PROGRAM MAIN
VAR
	bStart 						: BOOL;
	bEnable 					: BOOL;
	bDisable 					: BOOL;
	bReset 						: BOOL;
	bStop						: BOOL;
	nCase 						: UINT;
	nDemoSequenceState			: UINT;
	
	fbMover						: MC_PlanarMover;
	cmdFB						: MC_PlanarFeedback;
	stMoverState				: MC_PLANAR_STATE;
	stMoverPosition				: ARRAY[1..5] OF PositionXYC;
	fbDnyMove					: DynamicConstraint_PathXY;
	fbDnyRotate					: DynamicConstraint_Coordinates;
	stMoveCOptions				: ST_MoveCOptions;
	
	// Homing
	fbHomeATasks				: FB_TaskMoveA_tilt(fbMover := fbMover);
	fbHomeBTasks				: FB_TaskMoveB_tilt(fbMover := fbMover);
	fbHomeZTasks				: FB_TaskMoveZ(fbMover := fbMover);
	fbHomeCTasks				: FB_TaskMoveC(fbMover := fbMover);
	fbHomeToPositionTasks		: FB_TaskMoveToPosition(fbMover := fbMover);
	fb_home_sequence			: bajp_jobmgmt.FB_QueueJobContainer;
	fb_home_job					: bajp_jobmgmt.FB_Executor;
	
	// Demo Pattern
	fbMoveToPositionTasks		: ARRAY [1..9] OF FB_TaskMoveToPosition(fbMover := fbMover);
	fbMoveCTasks				: ARRAY [1..5] OF FB_TaskMoveC(fbMover := fbMover);
	fbMoveZTasks				: ARRAY [1..2] OF FB_TaskMoveZ(fbMover := fbMover);
	fbMoveATasks				: ARRAY [1..3] OF FB_TaskMoveA_tilt(fbMover := fbMover);
	fbMoveBTasks				: ARRAY [1..3] OF FB_TaskMoveB_tilt(fbMover := fbMover);
	fbMoveAB_ATasks				: ARRAY [1..3] OF FB_TaskMoveA_tilt(fbMover := fbMover);
	fbMoveAB_BTasks				: ARRAY [1..3] OF FB_TaskMoveB_tilt(fbMover := fbMover);
	fbMoveZTask_init			: FB_TaskMoveZ(fbMover := fbMover);
	
	fb_positioning_job			: bajp_jobmgmt.FB_BatchJobContainer;
	fb_rotation_job				: bajp_jobmgmt.FB_BatchJobContainer;
	fb_vertical_repeat_jobs		: bajp_jobmgmt.FB_BatchJobContainer;
	fb_tilt_A_repeat_jobs		: bajp_jobmgmt.FB_BatchJobContainer;
	fb_tilt_B_repeat_jobs		: bajp_jobmgmt.FB_BatchJobContainer;
	fb_tilt_AB_cycle_jobs		: bajp_jobmgmt.FB_BatchJobContainer;
	fb_demo_job					: bajp_jobmgmt.FB_BatchJobContainer;
	fb_manu_job					: bajp_jobmgmt.FB_QueueJobContainer;
	fbJob						: bajp_jobmgmt.FB_Executor;
	i: UINT;
	current_action : STRING;
	manual_command: iManualCommand;
	
	//試運転用パラメーター      
	(*          			
	Vel							: UDINT	:= 100;
	Acc							: UDINT	:= 1000;
	Dcc							: UDINT	:= 1000;
	Jerk						: UDINT	:= 5000;
	Ang_Vel						: UDINT	:= 100;
	Ang_Acc						: UDINT	:= 1000;
	Ang_Dcc						: UDINT	:= 1000;
	Ang_Jerk					: UDINT	:= 5000;
	*)             			
	 //デモ用パラメーター               			
	              			
	Vel							: UDINT	:= 400;
	Acc							: UDINT	:= 4000;
	Dcc							: UDINT	:= 4000;
	Jerk						: UDINT	:= 20000;
	Ang_Vel						: UDINT	:= 360;
	Ang_Acc						: UDINT	:= 3600;
	Ang_Dcc						: UDINT	:= 3600;
	Ang_Jerk					: UDINT	:= 36000;
	              			
	                			
	Height						: LREAL	:= 2.0;
	Cnt							: UINT;
	Z_High						: LREAL := 6.0;
	Z_Low						: LREAL := 2.0;
	A_Tilt						: LREAL := 0.0;
	B_Tilt						: LREAL := 0.0;
	Tilt						: LREAL := 2.5;
	Rotaion_Ang					: LREAL := 1.5;
	Estop						: BOOL;
	StopStep					: INT;
	fbDnyMoveEstop				: DynamicConstraint_PathXY;
	RotaionBit					: BOOL;
	Init_Angle					: BOOL;
	Init_Height_Tilt			: BOOL;
	
	Height_Tilt_Recover_Step	: INT;
	Init_Angle_Step				: INT;
	
	//  Utility Initial  -----------------------------------
	fbENviroment				: FB_TcIoXPlanarEnvironment;
	fbVisuXpalnar				: FB_XPlanarUtilityVisu;
	ipXpu						: I_TcIoXPlanarProcessingUnit;
	                			
	fbTcIoMover					: FB_TcIoXPlanarMover;
	ipXpm						: I_TcIoXPlanarMover;
	ipXpmsa						: I_XPlanarMoverScopeAdr;
	                			
	nStateInitXpu				: INT;
	bInit						: BOOL := FALSE;

	LampTimer					: TON;
	ServoON						: BOOL;
	Error						: BOOL;
	Init_Start					: BOOL;

	
	Manupilate_Start: BOOL;
	nManupilationState: UINT;
	nJobConfigState: INT;
	Demo_Start: BOOL;
	manu_mode: BOOL;
	manual_command_event: BOOL;
	manual_command_event_mem: BOOL;
	manupilator_buttons: ARRAY [0..49] OF BOOL;
END_VAR

VAR CONSTANT
	INIT_STEP	:	INT	 	:= 0;
	INIT_TILT 	: 	LREAL 	:= 0.0;
	INIT_HEIGHT :	LREAL 	:= 3.0;
	
END_VAR

//初期動作
IF NOT bInit THEN
		CASE nStateInitXpu OF
			0://Utilityの有効化
				IF fbENviroment.Init(TRUE) THEN
					fbENviroment.Init(FALSE);
					nStateInitXpu:=1;
				END_IF
			1://Utilityの実行を確認
				ipXpu:=fbENviroment.XpuTcIo(1);
				
				IF ipXpu<>0 THEN
					nStateInitXpu:=2;
				END_IF
				
			2://Job生成
				bInit := TRUE;
		END_CASE
	RETURN;
END_IF


fbMover.Update();
cmdFB.Update();
ACT_Lamp_Ctrl();
stMoverState 					:= fbMover.MCTOPLC.STD.State;

//サーボオン
IF bEnable THEN
	fbMover.Enable(cmdFB);
	bEnable := FALSE;
END_IF

//サーボオフ
IF bDisable THEN
	fbMover.Disable(cmdFB);
	nDemoSequenceState := 0;
	nManupilationState := 0;
	nCase := 0;
	IF fbjob.reset() THEN
		bDisable	:= FALSE;
	END_IF
END_IF

//サーボオン＋動作ステップが０番の時にデモ動作開始
IF stMoverState = MC_PLANAR_STATE.Enabled THEN
	IF Init_Start THEN
		// 原点復帰ボタンが押されたときの処理
		IF fb_manu_job.reset() THEN
			nCase 		:= 1;
			nManupilationState := 0;
			Init_Start	:= FALSE;
		END_IF
	END_IF
	CASE nManupilationState OF
		0: // 待機状態
			IF manu_mode AND nDemoSequenceState = 0 AND nCase = 5 THEN
				// Manual Modeボタンが押された時の処理
				nCase := 0;
				nManupilationState := 1;
			ELSE
				manu_mode := FALSE;
			END_IF
			// avoid
		1: // Clear jobs
			IF fbJob.reset() THEN
				IF manu_mode THEN
					MakeTasks();
					fb_manu_job.id := 'Manual';
					fbJob.future := fb_manu_job;
					nManupilationState := 2;
				ELSE
					nManupilationState := 0;
				END_IF
			END_IF
		2:// 非同期タスク発行
			manual_command_event := FALSE;
			FOR i := 0 TO 49 DO
				// HMIボタン入力
				IF manupilator_buttons[i] THEN
					manual_command_event := TRUE; // イベントフラグ
					manual_command.i_com := i; // コマンド番号をMenualCommand型のenumへ変換（UNION）
				END_IF
			END_FOR
		
			IF manual_command_event AND NOT manual_command_event_mem THEN
				// イベントフラグ立ち上がり条件の作成
				CASE manual_command.com OF
					// コマンド番号毎にタスクをキューに登録
					ManualCommand.move_pos_c1:
						fb_manu_job.add_future(fbMoveToPositionTasks[7]);
					ManualCommand.move_pos_c2:
						fb_manu_job.add_future(fbMoveToPositionTasks[1]);					
					ManualCommand.move_pos_c3:
						fb_manu_job.add_future(fbMoveToPositionTasks[8]);
					ManualCommand.move_pos_L1:
						fb_manu_job.add_future(fbMoveToPositionTasks[2]);	
					ManualCommand.move_pos_L2:
						fb_manu_job.add_future(fbMoveToPositionTasks[6]);
					ManualCommand.move_pos_L3:
						fb_manu_job.add_future(fbMoveToPositionTasks[3]);	
					ManualCommand.move_pos_r1:
						fb_manu_job.add_future(fbMoveToPositionTasks[4]);						
					ManualCommand.move_pos_r2:
						fb_manu_job.add_future(fbMoveToPositionTasks[9]);
					ManualCommand.move_pos_r3:
						fb_manu_job.add_future(fbMoveToPositionTasks[5]);						
					ManualCommand.move_roll_w:
						fb_manu_job.add_future(fbMoveCTasks[5]);
					ManualCommand.move_roll_n:
						fb_manu_job.add_future(fbMoveCTasks[1]);
					ManualCommand.move_roll_e:
						fb_manu_job.add_future(fbMoveCTasks[3]);
					ManualCommand.move_roll_s:
						fb_manu_job.add_future(fbMoveCTasks[4]);
					ManualCommand.move_tilt_up_front:
						fb_manu_job.add_future(fbMoveATasks[1]);					
					ManualCommand.move_tilt_up_left:
						fb_manu_job.add_future(fbMoveATasks[2]);					
					ManualCommand.move_tilt_up_rear:
						fb_manu_job.add_future(fbMoveBTasks[1]);					
					ManualCommand.move_tilt_up_right:
						fb_manu_job.add_future(fbMoveBTasks[2]);
					ManualCommand.move_tilt_horizontal:
						fb_manu_job.add_future(fbMoveATasks[3]);
						fb_manu_job.add_future(fbMoveBTasks[3]);
					ManualCommand.move_up:
						fb_manu_job.add_future(fbMoveZTasks[1]);
					ManualCommand.move_down:					
						fb_manu_job.add_future(fbMoveZTasks[2]);
				END_CASE
			END_IF
			manual_command_event_mem := manual_command_event;
			//実行
			IF fbJob.current_state = bajp_jobmgmt.E_FutureExecutionState.wait_for_process AND fbJob.ready THEN
				fbJob.start();
			END_IF
			IF fbJob.execute() AND fbJob.nErrorID = 0 THEN
				fbJob.init();
			END_IF
			//停止動作
			IF bStop THEN
				fbJob.abort();	
			END_IF
			
			IF bReset THEN
				fbJob.start();
			END_IF
			current_action := fbJob.active_future_id;
			IF NOT manu_mode THEN
				nManupilationState := 1;
			END_IF
	END_CASE
END_IF


//原点復帰
CASE nCase OF
	0:
		// avoid step
		
	1: // Clear jobs
		nDemoSequenceState := 0;
		// それまで行われいたfbJobとfb_home_jobをクリアする。（数サイクル要する）
		IF fbJob.reset() THEN
			IF fb_home_job.reset() THEN
				nCase := 2;
			END_IF			
		END_IF
	2: // 原点復帰ジョブの組み立て。1サイクルだけ実行しなければならない。
		MakeJob_Home();
		fb_home_sequence.id := 'Initiliaze';
		fb_home_sequence.add_future(fbHomeATasks);
		fb_home_sequence.add_future(fbHomeBTasks);
		fb_home_sequence.add_future(fbHomeZTasks);
		fb_home_sequence.add_future(fbHomeCTasks);
		fb_home_job.future := fb_home_sequence;
		IF fb_home_job.init() THEN
			nCase := 3;
		END_IF
	3: // execute initialization
		IF fb_home_job.current_state = bajp_jobmgmt.E_FutureExecutionState.wait_for_process AND fb_home_job.ready THEN
			fb_home_job.start();
		END_IF
		IF fb_home_job.execute() AND fb_home_job.nErrorID = 0 THEN
			nCase := 4;
		END_IF
		//停止動作
		IF bStop THEN
			fb_home_job.abort();	
		END_IF
		
		IF bReset THEN
			fb_home_job.start();
		END_IF
		current_action := fb_home_job.active_future_id;
	4: // Job creating.
		// Container クラスのreset()メソッドで子要素もリセットできるので、一括リセットするため、いったん全てのコンテナツリーをfb_demo_jobに登録する
		fb_demo_job.add_future(fb_positioning_job);
		fb_demo_job.add_future(fb_rotation_job);
		fb_demo_job.add_future(fb_vertical_repeat_jobs);
		fb_demo_job.add_future(fb_tilt_A_repeat_jobs);
		fb_demo_job.add_future(fb_tilt_B_repeat_jobs);
		fb_demo_job.add_future(fb_tilt_AB_cycle_jobs);
		fb_demo_job.add_future(fbMoveZTask_init);
		IF fb_demo_job.reset() THEN
			// リセットを実行し、完了後、再度ジョブをコンテナに登録する
			// リセットによってジョブ、タスク間の関係さえも切れてしまう。
			// よって、2度手間だがリセットのためにジョブモデル構築し、もう一度ジョブモデルを構築しなおす必要がある。
			// どの状態で終了したかわからない原点復帰ではこの処理が必要。
			MakeJob_DemoPattern();
			fb_demo_job.id := 'Demo';
			fb_demo_job.add_future(fb_positioning_job);
			fb_demo_job.add_future(fb_rotation_job);
			fb_demo_job.add_future(fb_vertical_repeat_jobs);
			fb_demo_job.add_future(fb_tilt_A_repeat_jobs);
			fb_demo_job.add_future(fb_tilt_B_repeat_jobs);
			fb_demo_job.add_future(fb_tilt_AB_cycle_jobs);
			fb_demo_job.add_future(fbMoveZTask_init);
			nCase := 5;
		END_IF
	5: // Ready to start
		IF stMoverState = MC_PLANAR_STATE.Disabled THEN
			nCase := 0;
			nDemoSequenceState := 0;
		END_IF
END_CASE


//デモ動作開始
IF Demo_Start THEN
	IF nCase = 5 AND nDemoSequenceState = 0 THEN
		nDemoSequenceState 		:= 1;
	END_IF
	Demo_Start	:= FALSE;	
END_IF


// デモ動作
CASE nDemoSequenceState OF
	0:
		// avoid
	1:
		fbJob.future := fb_demo_job;
		MakeTasks();
		// 初期化
		IF fbJob.init() THEN
			nDemoSequenceState := 2;
		END_IF
	2:
		//デモモード実行
		IF fbJob.current_state = bajp_jobmgmt.E_FutureExecutionState.wait_for_process AND fbJob.ready THEN
			fbJob.start();
		END_IF
		IF fbJob.execute() AND fbJob.nErrorID = 0 THEN
			nDemoSequenceState := 1;
		END_IF
		//停止動作
		IF bStop THEN
			fbJob.abort();	
		END_IF
		
		IF bReset THEN
			fbJob.start();
		END_IF
		current_action := fbJob.active_future_id;
END_CASE

IF bStop THEN
	bStop		:= FALSE;
END_IF


//動作とエラーリセット
IF bReset THEN
	fbMover.Reset(cmdFB);
	bReset		:= FALSE;
END_IF

IoT();

ACTION ACT_Lamp_Ctrl:
Error := FALSE;

IF stMoverState = MC_PLANAR_STATE.Disabled THEN
	LampTimer.IN := NOT LampTimer.Q;
	LampTimer.PT := T#750MS;
	LampTimer();
	
	IF LampTimer.Q THEN
		ServoON := NOT ServoON;
		
	END_IF
ELSIF stMoverState = MC_PLANAR_STATE.Enabled THEN	
	ServoON := TRUE;

	
ELSIF stMoverState = MC_PLANAR_STATE.Error THEN	
	Error := TRUE;

END_IF
END_ACTION

METHOD MakeJob_DemoPattern : BOOL
VAR_INPUT
END_VAR

// 直線動作タスク追加
FOR i := 1 TO 5 DO
	fb_positioning_job.add_future(fbMoveToPositionTasks[i]);
END_FOR
fb_positioning_job.add_future(fbMoveToPositionTasks[1]);

// 回転動作タスク追加
FOR i := 1 TO  2 DO
	fb_rotation_job.add_future(fbMoveCTasks[i]);
END_FOR

// 上下動作タスク追加
FOR i := 1 TO 9 DO
	fb_vertical_repeat_jobs.add_future(fbMoveZTasks[1]); //MAX_TASKが10までなので前後半配列に分けて登録
	fb_vertical_repeat_jobs.add_future(fbMoveZTasks[2]);
END_FOR

fb_vertical_repeat_jobs.add_future(fbMoveZTasks[1]);

// 傾きA動作タスク追加
FOR i := 1 TO 10 DO
	fb_tilt_A_repeat_jobs.add_future(fbMoveATasks[1]);
	IF i = 10 THEN
		fb_tilt_A_repeat_jobs.add_future(fbMoveATasks[3]);
	ELSE
		fb_tilt_A_repeat_jobs.add_future(fbMoveATasks[2]);
	END_IF
END_FOR

// 傾きB動作タスク追加
FOR i := 1 TO 10 DO
	fb_tilt_B_repeat_jobs.add_future(fbMoveBTasks[1]);
	IF i = 10 THEN
		fb_tilt_B_repeat_jobs.add_future(fbMoveBTasks[3]);
	ELSE
		fb_tilt_B_repeat_jobs.add_future(fbMoveBTasks[2]);
	END_IF
END_FOR

// AB両方の傾き
FOR i := 1 TO 4 DO
	fb_tilt_AB_cycle_jobs.add_future(fbMoveAB_ATasks[1]);
	fb_tilt_AB_cycle_jobs.add_future(fbMoveAB_BTasks[1]);
	fb_tilt_AB_cycle_jobs.add_future(fbMoveAB_ATasks[2]);
	fb_tilt_AB_cycle_jobs.add_future(fbMoveAB_BTasks[2]);
END_FOR
fb_tilt_AB_cycle_jobs.add_future(fbMoveAB_ATasks[3]);
fb_tilt_AB_cycle_jobs.add_future(fbMoveAB_BTasks[3]);

MakeJob_DemoPattern := TRUE;
END_METHOD

ACTION MakeJob_Home:
IF fb_home_job.init() THEN
	fbHomeATasks.set_target_position(0);
	fbHomeATasks.set_dynamics(Vel, Acc, Dcc, Jerk);
	fbHomeBTasks.set_target_position(0);
	fbHomeBTasks.set_dynamics(Vel, Acc, Dcc, Jerk);
	fbHomeZTasks.set_target_position(INIT_HEIGHT);
	fbHomeZTasks.set_dynamics(Vel, Acc, Dcc, Jerk);
	fbHomeCTasks.set_target_position(0);
	fbHomeCTasks.set_dynamics(Coord_Mcs_C1,Ang_Vel,Ang_Acc,Ang_Dcc,Ang_Jerk);
	//fbHomeToPositionTasks.set_target_position(240,120,0);
	//fbHomeToPositionTasks.set_dynamics(Vel, Acc, Dcc, Jerk);
END_IF
END_ACTION

METHOD MakeTasks : BOOL
VAR_INPUT
END_VAR

// 直線動作タスク追加
fbMoveToPositionTasks[1].set_target_position(240,120,0);
fbMoveToPositionTasks[2].set_target_position(80,80,0);
fbMoveToPositionTasks[3].set_target_position(80,160,0);
fbMoveToPositionTasks[4].set_target_position(400,160,0);
fbMoveToPositionTasks[5].set_target_position(400,80,0);
fbMoveToPositionTasks[6].set_target_position(80,120,0);
fbMoveToPositionTasks[7].set_target_position(240,80,0);
fbMoveToPositionTasks[8].set_target_position(240,160,0);
fbMoveToPositionTasks[9].set_target_position(400,120,0);
FOR i := 1 TO 9 DO
	fbMoveToPositionTasks[i].set_dynamics(Vel, Acc, Dcc, Jerk);
END_FOR

// 回転動作タスク追加
fbMoveCTasks[1].set_target_position(0.0);
fbMoveCTasks[2].set_target_position(360.0);
fbMoveCTasks[3].set_target_position(90.0);
fbMoveCTasks[4].set_target_position(180.0);
fbMoveCTasks[5].set_target_position(270.0);
FOR i := 1 TO  5 DO
	fbMoveCTasks[i].set_dynamics(Coord_Mcs_C1,Ang_Vel,Ang_Acc,Ang_Dcc,Ang_Jerk);
END_FOR

// 上下動作タスク追加
fbMoveZTasks[1].set_target_position(Z_High);
fbMoveZTasks[1].set_dynamics(Vel, Acc, Dcc, Jerk);
fbMoveZTasks[2].set_target_position(Z_Low);
fbMoveZTasks[2].set_dynamics(Vel, Acc, Dcc, Jerk);

// 傾きA動作タスク追加
fbMoveATasks[1].set_target_position(Tilt);
fbMoveATasks[1].set_dynamics(Vel, Acc, Dcc, Jerk);
fbMoveATasks[2].set_target_position(-Tilt);
fbMoveATasks[2].set_dynamics(Vel, Acc, Dcc, Jerk);
fbMoveATasks[3].set_target_position(0);
fbMoveATasks[3].set_dynamics(Vel, Acc, Dcc, Jerk);

// 傾きB動作タスク追加
fbMoveBTasks[1].set_target_position(Tilt);
fbMoveBTasks[1].set_dynamics(Vel, Acc, Dcc, Jerk);
fbMoveBTasks[2].set_target_position(0 - Tilt);
fbMoveBTasks[2].set_dynamics(Vel, Acc, Dcc, Jerk);
fbMoveBTasks[3].set_target_position(0);
fbMoveBTasks[3].set_dynamics(Vel, Acc, Dcc, Jerk);

// AB両方の傾き
fbMoveAB_ATasks[1].set_target_position(Rotaion_Ang);
fbMoveAB_ATasks[1].set_dynamics(Vel, Acc, Dcc, Jerk);
fbMoveAB_ATasks[2].set_target_position(-Rotaion_Ang);
fbMoveAB_ATasks[2].set_dynamics(Vel, Acc, Dcc, Jerk);
fbMoveAB_ATasks[3].set_target_position(0);
fbMoveAB_ATasks[3].set_dynamics(Vel, Acc, Dcc, Jerk);
fbMoveAB_BTasks[1].set_target_position(Rotaion_Ang);
fbMoveAB_BTasks[1].set_dynamics(Vel, Acc, Dcc, Jerk);
fbMoveAB_BTasks[2].set_target_position(-Rotaion_Ang);
fbMoveAB_BTasks[2].set_dynamics(Vel, Acc, Dcc, Jerk);
fbMoveAB_BTasks[3].set_target_position(0);
fbMoveAB_BTasks[3].set_dynamics(Vel, Acc, Dcc, Jerk);

// 初期状態高さへ戻る
fbMoveZTask_init.set_target_position(INIT_HEIGHT);
fbMoveZTask_init.set_dynamics(Vel, Acc, Dcc, Jerk);
END_METHOD

END_PROGRAM

(* stored: Version 1.1.0.1, ProductVersion 3.1.4024.12
   POU MAIN: Id {09544d0d-3edc-4a61-aaa2-1eeba1575761}, SpecialFunc None
   Action ACT_Lamp_Ctrl: Id {f67b75e7-2e3d-4471-91f9-9d6b1ed7fc89}
   Method MakeJob_DemoPattern: Id {5c1d0e90-5dce-4289-b8a5-8f97c2323b70}
   Action MakeJob_Home: Id {af803ab2-5260-4545-8bd1-989c6b0d6468}
   Method MakeTasks: Id {c18f96ce-3a73-48c3-89c6-3367fd26b018} *)
